// TwinCAT 3 PLC project HomePLC_Logging
// Title: HomePLC Logging
// Company: Tom Oyen
// Author: Tom Oyen
// ProjectVersion: 1.0.1
// Description: Logging
// ProgramVersion: 3.1.4024.0
// libraries:
//   Tc2_Standard, * (Beckhoff Automation GmbH)
//   Tc2_System, * (Beckhoff Automation GmbH)
//   Tc3_EventLogger, * (Beckhoff Automation GmbH)
//   Tc3_Module, * (Beckhoff Automation GmbH)
// project tree:
//   / PlcTask.TcTTO
//   POUs/ class_Tc3Eventlogger.TcPOU, E_MessageType.TcTLEO, LogMessage.TcPOU
//   Project Information/ F_GetCompany.TcPOU, F_GetTitle.TcPOU, F_GetVersion.TcPOU
//   Version/ Global_Version.TcGVL

CONFIGURATION HomePLC_Logging
    RESOURCE PLC ON TwinCAT3
        TASK PlcTask(INTERVAL := T#10ms, PRIORITY := 20);
    END_RESOURCE
END_CONFIGURATION

// ---- POUs/E_MessageType.TcTLEO
{attribute 'qualified_only'}
{attribute 'strict'}
TYPE E_MessageType :
(
	Hint	:= 1,
	Warn	:= 2,
	Error	:= 4
) DWORD;
END_TYPE

// ADSLOG_MSGTYPE_HINT = 1: Message type is hint.
// ADSLOG_MSGTYPE_WARN = 2: Message type is warning.
// ADSLOG_MSGTYPE_ERROR = 4: Message type is error.

// ---- Version/Global_Version.TcGVL
{attribute 'TcGenerated'}
{attribute 'no-analysis'}
{attribute 'linkalways'}
// This function has been automatically generated from the project information.
VAR_GLOBAL CONSTANT
	{attribute 'const_non_replaced'}
	stLibVersion_HomePLC_Logging : ST_LibVersion := (iMajor := 1, iMinor := 0, iBuild := 1, iRevision := 0, nFlags := 0, sVersion := '1.0.1');
END_VAR

// ---- POUs/class_Tc3Eventlogger.TcPOU
// Event logger based on the TC3 Eventlogger
FUNCTION_BLOCK class_Tc3Eventlogger
VAR
	fbMessageVerbose		: FB_TcMessage;		// Verbose message, e.g. for debugging
	fbMessageInfo			: FB_TcMessage;		// Info message, e.g. for event logging
	fbMessageWarning		: FB_TcMessage;		// Warning message
	fbMessageError			: FB_TcMessage;		// Error message
	hrLastError				: HRESULT;			// Last error when sending a message
	
	bEnableVerbose			: BOOL;				// Enable verbose messages
END_VAR

// In order to use this FB, an event class named "Eventlogger" needs to be created under SYSTEM/Type System/Event classes
// The event class needs to have two events:
// - Name: VerboseEvent, Display Text: {0}, Severity: Verbose
// - Name: InfoEvent, Display Text: {0}, Severity: Info

// Add a debug message (verbose)
METHOD AddDebug : BOOL
VAR_INPUT
	Message		: STRING;			// Message to log
END_VAR
VAR
	hr			: HRESULT;			// Result of sending the message
END_VAR
IF bEnableVerbose THEN
	// Add input message to arguments
	fbMessageVerbose.ipArguments.Clear().AddString(Message);
	
	// Send message
	hr := fbMessageVerbose.Send(0);
	
	// Check if send failed
	IF FAILED(hr) THEN
		// Store last error
		hrLastError := hr;
	END_IF
END_IF
END_METHOD

// Add an info message
METHOD AddError : BOOL
VAR_INPUT
	Message		: STRING;			// Message to log
END_VAR
VAR
	hr			: HRESULT;			// Result of sending the message
END_VAR
// Add input message to arguments
fbMessageError.ipArguments.Clear().AddString(Message);

// Send message
hr := fbMessageError.Send(0);

// Check if send failed
IF FAILED(hr) THEN
	// Store last error
	hrLastError := hr;
END_IF
END_METHOD

// Add an info message
METHOD AddInfo : BOOL
VAR_INPUT
	Message		: STRING;			// Message to log
END_VAR
VAR
	hr			: HRESULT;			// Result of sending the message
END_VAR
// Add input message to arguments
fbMessageInfo.ipArguments.Clear().AddString(Message);

// Send message
hr := fbMessageInfo.Send(0);

// Check if send failed
IF FAILED(hr) THEN
	// Store last error
	hrLastError := hr;
END_IF
END_METHOD

// Add an info message
METHOD AddWarning : BOOL
VAR_INPUT
	Message		: STRING;			// Message to log
END_VAR
VAR
	hr			: HRESULT;			// Result of sending the message
END_VAR
// Add input message to arguments
fbMessageWarning.ipArguments.Clear().AddString(Message);

// Send message
hr := fbMessageWarning.Send(0);

// Check if send failed
IF FAILED(hr) THEN
	// Store last error
	hrLastError := hr;
END_IF
END_METHOD

// Initialize the logger
METHOD Init : BOOL
VAR_INPUT
	sSource			: STRING;					// Name to be used as the source of the messages
	bEnableVerbose	: BOOL;						// Enable verbose messages
END_VAR
VAR
	fbSourceInfo	: FB_TcSourceInfo;			// Source info
END_VAR
// Set source
fbSourceInfo.Clear();
fbSourceInfo.sName := sSource;

// Create messages
fbMessageVerbose.CreateEx(TC_EVENTS.EventLogger.VerboseEvent, fbSourceInfo);
fbMessageInfo.CreateEx(TC_EVENTS.EventLogger.InfoEvent, fbSourceInfo);
fbMessageWarning.CreateEx(TC_EVENTS.EventLogger.WarningEvent, fbSourceInfo);
fbMessageError.CreateEx(TC_EVENTS.EventLogger.ErrorEvent, fbSourceInfo);

// Enable/disable logging
THIS^.bEnableVerbose := bEnableVerbose;
END_METHOD

END_FUNCTION_BLOCK

// ---- POUs/LogMessage.TcPOU
FUNCTION LogMessage : BOOL
VAR_INPUT
	sLogMessage		: STRING[255];			// String size set to 255, default is 80
	eType			: E_MessageType;
END_VAR

// ADSLOG_MSGTYPE_HINT: Message type is hint.
// ADSLOG_MSGTYPE_WARN: Message type is warning.
// ADSLOG_MSGTYPE_ERROR: Message type is error.
// ADSLOG_MSGTYPE_LOG: Message is written into the LOG.
// ADSLOG_MSGTYPE_MSGBOX: Message is output to a message box. Caution: This functionality is not available under Windows CE.
// ADSLOG_MSGTYPE_STRING: Message is a directly given STRING (default).

ADSLOGSTR(eType OR ADSLOG_MSGTYPE_LOG, sLogMessage, '');

END_FUNCTION

// ---- Project Information/F_GetCompany.TcPOU
// This function has been automatically generated from the project information.
{attribute 'signature_flag' := '1073741824'}
{attribute 'TcGenerated'}
{attribute 'no-analysis'}
FUNCTION F_GetCompany : WSTRING
VAR_INPUT
	
END_VAR

F_GetCompany := "Tom Oyen";

END_FUNCTION

// ---- Project Information/F_GetTitle.TcPOU
// This function has been automatically generated from the project information.
{attribute 'signature_flag' := '1073741824'}
{attribute 'TcGenerated'}
{attribute 'no-analysis'}
FUNCTION F_GetTitle : WSTRING
VAR_INPUT
	
END_VAR

F_GetTitle := "HomePLC Logging";

END_FUNCTION

// ---- Project Information/F_GetVersion.TcPOU
// This function has been automatically generated from the project information.
{attribute 'signature_flag' := '1073741824'}
{attribute 'TcGenerated'}
{attribute 'no-analysis'}
FUNCTION F_GetVersion : ST_LibVersion
VAR_INPUT
	
END_VAR

F_GetVersion.iMajor := 1;
F_GetVersion.iMinor := 0;
F_GetVersion.iBuild := 1;
F_GetVersion.iRevision := 0;
F_GetVersion.sVersion := '1.0.1';
F_GetVersion.nFlags := 0;

END_FUNCTION
